INTERFACE FuzzyInferenceSystem

METHOD Defuzzification :REAL;
VAR_INPUT
END_VAR
END_METHOD

METHOD Fuzzyfication 
VAR_INPUT
END_VAR
END_METHOD

END_INTERFACE

(* stored: Version 1.1.0.1, ProductVersion 3.1.4024.6
   Itf FuzzyInferenceSystem: Id {d92d4760-a7db-4f60-8cab-24390dffeeed}
   Method Defuzzification: Id {968ac9b4-797b-494e-af6b-5cf639dc62e2}
   Method Fuzzyfication: Id {1ae2ebed-eef4-413d-bf5b-2cc292ccedf5} *)
